// TIA Portal V16 export
// export: Created 2024-09-05T17:39:13.0311728Z, ExportSetting WithDefaults, DisplayName Totally Integrated Automation Portal, DisplayVersion V16 Update 6, DisplayName TIA Portal Version Control Interface, DisplayVersion V16 Update 2, DisplayName TIA Portal Openness, DisplayVersion V16 Update 6, DisplayName STEP 7 Professional, DisplayVersion V16 Update 6, DisplayName STEP 7 Safety, DisplayVersion V16, DisplayName WinCC Advanced, DisplayVersion V16 Update 6
DATA_BLOCK "Manipulator_main_DB"   // DB42
VERSION : 0.1
// stored: AutoNumber true, DBAccessibleFromOPCUA true, InstanceOfName Manipulator_main, InstanceOfType FB
"Manipulator_main"
   // VAR
   //    PUT_Instance : PUT;
   //    GET_Instance : GET;
   //    GetStatusMem : Word;
   //    PutStatusMem : Word;
   //    GetCounterNDR : ULInt;
   //    PutCounterDone : ULInt;
   //    GetCounterNDR_last : ULInt;
   //    PutCounterDone_last : ULInt;
   //    GetCommOK : Bool;
   //    PutCommOK : Bool;
   //    R_TRIG_GetNDR : R_TRIG;
   //    R_TRIG_PutDone : R_TRIG;
   //    IEC_Timer_GetCommOK { S7_SetPoint := 'True'} : TOF_TIME;
   //    IEC_Timer_PutCommOK { S7_SetPoint := 'True'} : TOF_TIME;
   // END_VAR
BEGIN
END_DATA_BLOCK
